FUNCTION F_TargetWindowReached : BOOL
VAR_INPUT
	fCurrentPos: LREAL;
	fTargetPos: LREAL;
	fWindow: LREAL;
END_VAR


F_TargetWindowReached := fCurrentPos >= (fTargetPos - fWindow) AND fCurrentPos <= (fTargetPos + fWindow);

END_FUNCTION

(* stored: Version 1.1.0.1, ProductVersion 3.1.4020.12
   POU F_TargetWindowReached: Id {a1d9bfbe-a94d-4f6b-92e3-d1d03203f03c}, SpecialFunc None *)
